{attribute 'no_explicit_call' := 'do not call this POU directly'}
FUNCTION_BLOCK FINAL FB_LoggedEventsSortDescending IMPLEMENTS I_LoggedEventsSort
VAR_INPUT
END_VAR
VAR_OUTPUT
END_VAR
VAR
END_VAR

METHOD PRIVATE GetLastIndex : UDINT
VAR_IN_OUT
	aLoggedEvents	: T_LoggedEvents;
END_VAR

VAR
	i 				: UDINT;
	nLastIndex		: UDINT;
	stLoggedEvent 	: ST_LoggedEvent;
END_VAR
FOR i := 0 TO Param_EventLoggerListener.cMaxConcurrentEvents - 1 BY 1 DO
	IF aLoggedEvents[i].nUniqueId > 0 OR_ELSE aLoggedEvents[i].nSourceId > 0 THEN
		GetLastIndex := i;
	ELSE
		EXIT;
	END_IF
END_FOR;
END_METHOD

METHOD Sort : HRESULT
VAR_IN_OUT
	aLoggedEvents	: T_LoggedEvents;
END_VAR

VAR
	i 				: UDINT;
	nLastIndex		: UDINT;
	stTmpEvent 		: ST_LoggedEvent;
END_VAR
nLastIndex := GetLastIndex(aLoggedEvents);
IF nLastIndex = 0 THEN
	Sort := S_FALSE;
	RETURN;
END_IF

FOR i := nLastIndex TO (nLastIndex / 2) + 1 BY -1 DO
	MEMMOVE(destAddr:= ADR(stTmpEvent), srcAddr:= ADR(aLoggedEvents[i]), n:= SIZEOF(stTmpEvent)); 
	MEMMOVE(destAddr:= ADR(aLoggedEvents[i]), srcAddr:= ADR(aLoggedEvents[nLastIndex - i]), n:= SIZEOF(aLoggedEvents[i])); 
	MEMMOVE(destAddr:= ADR(aLoggedEvents[nLastIndex - i]), srcAddr:= ADR(stTmpEvent), n:= SIZEOF(stTmpEvent)); 
END_FOR

Sort := S_OK;
END_METHOD

END_FUNCTION_BLOCK

(* stored: Version 1.1.0.1, ProductVersion 3.1.4024.12
   POU FB_LoggedEventsSortDescending: Id {52712f22-095f-4017-8c07-06b74336489a}, SpecialFunc None
   Method GetLastIndex: Id {49c1ac21-d879-4770-9208-e6856db53834}
   Method Sort: Id {17a4d191-9b1c-4d74-8fbe-b1139cff1151} *)
